FUNCTION_BLOCK EL5042
VAR
	_io : EL5042_Data;
	{attribute addProperty Name "WcState"}
	_wcState : WcStateInputToggle;
	{attribute addProperty Name "Info data"}
	_infoData : InfoDataAdsDC;
END_VAR

PROPERTY IO : REFERENCE TO EL5042_Data
GET
IO REF= _io;
END_GET
END_PROPERTY

PROPERTY WcState : REFERENCE TO WcStateInputToggle
GET
WcState REF= _wcState;
END_GET
END_PROPERTY

END_FUNCTION_BLOCK

(* stored: Version 1.1.0.1, ProductVersion 3.1.4024.9
   POU EL5042: Id {f56e4a12-45e7-0bc6-254b-53af4cf813d1}, SpecialFunc None
   Property IO: Id {f04cc0ee-2c0f-0288-296b-b45d11b2510c}
   Get Get: Id {e26cb4f0-fc04-0f92-0817-25becadf0758}
   Property WcState: Id {2af59a99-e492-0af1-2a20-046505a46250}
   Get Get: Id {5aa8433b-3664-0364-254d-be24b0a5eb92} *)
